// TIA Portal V20 export
DATA_BLOCK "GLOBAL_PROCESS_COMP_HMI_IF_DB"   // DB212
{ S7_Optimized_Access := 'TRUE' }
// stored: AutoNumber false, MemoryReserve 100
   VAR
      PROCESS_COMP { S7_SetPoint := 'True'} : Array[0..20] of "MISC_PROCESS_COMP_HMI_UDT";
   END_VAR
BEGIN
   // PROCESS_COMP[0] : +ST010-TL01
   // PROCESS_COMP[1] : +ST010-TL02
   // PROCESS_COMP[2] : +ST020-TL01
   // PROCESS_COMP[3] : +ST020-TL02
   // PROCESS_COMP[4] : +ST020-TL01
   // PROCESS_COMP[5] : +ST020-TL09
   // PROCESS_COMP[6] : +ST020-TL10
   // PROCESS_COMP[7] : +ST020-TL12
   // PROCESS_COMP[10] : +ST025-TL01
   // PROCESS_COMP[11] : +ST025-TL02
   // PROCESS_COMP[12] : +ST030-TL01
   // PROCESS_COMP[13] : +ST030-TL03
   // PROCESS_COMP[14] : +ST030-TL04
   // PROCESS_COMP[15] : +ST020-CNV04
   // PROCESS_COMP[16] : +ST020-CNV05
   // PROCESS_COMP[17] : +ST020-CNV06
END_DATA_BLOCK
